FUNCTION_BLOCK FB_BaseComponent_HMI EXTENDS FB_BaseLoggerElement_HMI IMPLEMENTS ITF_BaseComponent_HMI
VAR
	itfBaseComponentConnector			: ITF_BaseComponent_HMI_Connector;
	refstBaseComponentDataHMI			: REFERENCE TO ST_BaseComponent_HMI;
END_VAR

END_FUNCTION_BLOCK

(* stored: Version 1.1.0.1
   POU FB_BaseComponent_HMI: Id {52a5d3de-74e5-09ff-1362-d8678f55ad3c}, SpecialFunc None *)
